RoboDK station: 2 - Pause.rdk

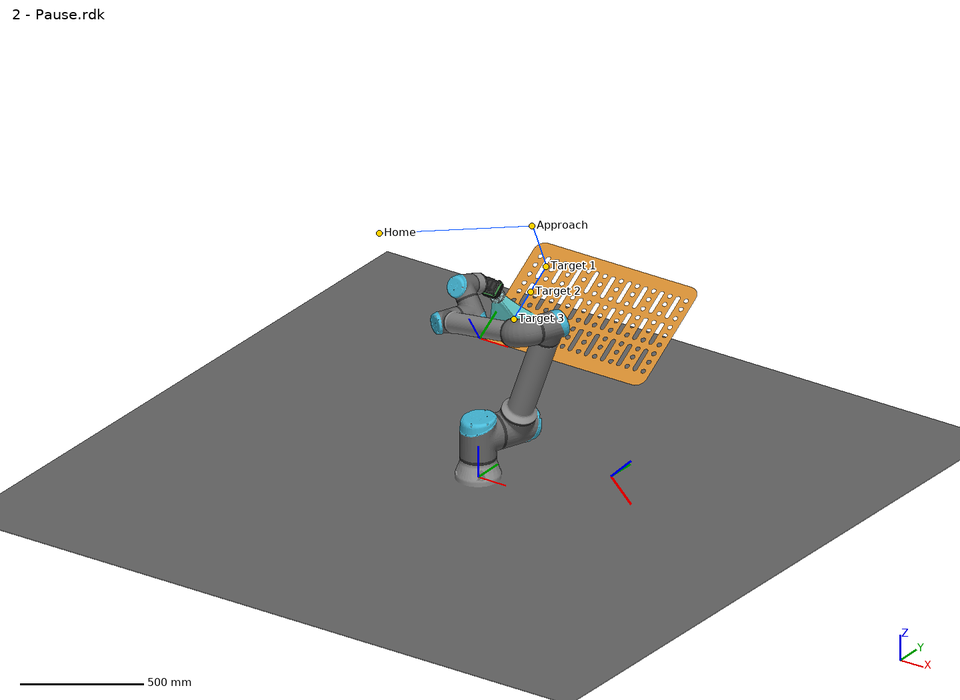
[picture v0: the station drawn from its stored meshes, robots at their saved joint values, targets as dots, program paths as lines]
Station 01B - Inspection_solved (saved by RoboDK 5.5.3). Poses are relative to the parent item; angles as X-Y-Z fixed-axis rotations.
Station parameters (name, value as stored): Palletizing Plugin
  - frame UR10e Base at (0, 0, 0) mm
    - robot UR10e: 6 axes, payload 10 kg, reach 1300 mm, repeatability 0.05 mm, weight 28.9 kg
        modified DH rows (alpha deg, a mm, theta deg, d mm): 0, 0, 0, 180.7; 90, 0, 180, 0; 0, 612.6, 0, 0; 0, 571.335, 0, 174.15; -90, 0, 0, 119.85; 90, 0, 180, 116.55
        joint limits [-360, -360, -360, -360, -360, -360] to [360, 360, 360, 360, 360, 360]; home [0, -90, -90, 0, 90, 0]; saved at [-200.514, -65.055, -131.307, -25.021, 26.504, -141.745]
      - tool Camera 2, TCP at (0, -175.95, 321.06) mm, rotated rx 40 ry 0 rz 0 deg, size 215.7 x 276.1 x 372.4 mm
  - frame Frame Inspection A at (-380.72, 555.26, 295.21) mm, rotated rx 32.84 ry 0 rz 0 deg
    - object Inspection A at (0, 0, 0) mm, size 800 x 500 x 0 mm, geometry from Inspection A.step
  - frame Frame Inspection B at (727.24, -100, 245.26) mm, rotated rx 0 ry 45.31 rz 0 deg
    - object Inspection B at (0, 0, 0) mm, size 202.5 x 1023.2 x 500 mm, geometry from Inspection B.step
  - frame World at (0, 0, 0) mm
    - object Floor at (0, 0, -7) mm, size 3000 x 3000 x 4.2 mm, geometry from Floor.step
    - target Target 1 (Cartesian target) at (-283.45, 884.6, 513.74) mm, rotated rx 147.16 ry 0 rz 180 deg; joints [135.813, -85.489, -103.576, -14.828, 46.752, 196.884] of UR10e
    - target Target 2 (Cartesian target) at (-284.92, 776.28, 443.82) mm, rotated rx 147.16 ry 0 rz 180 deg; joints [145.205, -76.522, -117.744, -14.151, 38.312, 203.004] of UR10e
    - target Target 3 (Cartesian target) at (-284.64, 658.67, 367.9) mm, rotated rx 147.16 ry 0 rz 180 deg; joints [159.486, -65.055, -131.307, -25.021, 26.504, 218.255] of UR10e
    - target Approach (Cartesian target) at (-305.13, 818.27, 718.21) mm, rotated rx 135.89 ry -14.46 rz 177.42 deg; joints [-214.79, -76.52, -99.79, -13.89, 34.11, -156.99] of UR10e
    - target Home (Cartesian target) at (-772.33, 407.48, 718.51) mm, rotated rx 135.87 ry -14.49 rz -140.85 deg; joints [-173.05, -76.51, -99.78, -13.89, 34.1, -156.98] of UR10e
  - program Prog1 (7 instructions, listed below)
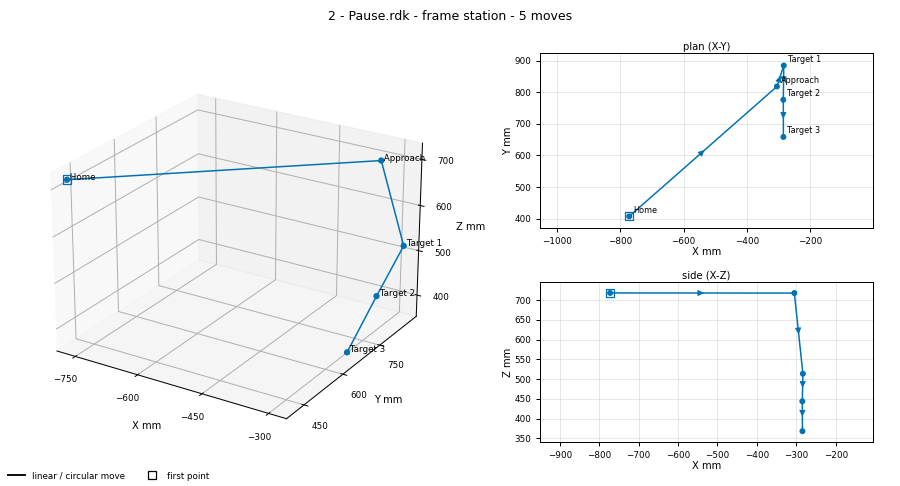
[picture p0: tool path of 2 - Pause.rdk in frame station, 5 of 5 moves have a stored position in this frame; points joined in program order, loops and branches not executed]

--- program Prog1 (robot UR10e) ---
  Set Ref.: World
  Set Tool: Camera 2
  MoveJ (Home)
  MoveL (Approach)
  MoveL (Target 1)
  MoveL (Target 2)
  MoveL (Target 3)
